{attribute 'qualified_only'}
VAR_GLOBAL
    logger          : LoggerADS;
END_VAR

(* stored: Version 1.1.0.1, ProductVersion 3.1.4026.18
   GVL GVL_Logger: Id {7cd63e60-a5dd-4b9b-a519-7d8c9472e8e8} *)
